Fanuc KAREL source: ko00053.KL

-- PROVISIONAL review KL for V1013-1; original PC SHA256 1e71e2e0424b7fda3cae7a66e169d6796f6002b1d3d6ba8bf153a4db3ede6087
-- Incomplete behavior may be omitted. Consult companion uncertainty JSON. Do not deploy.
PROGRAM KO00053
%NOLOCKGROUP
BEGIN
  -- UNRESOLVED_PC offsets 5-12; opcodes 9D,23
  -- UNRESOLVED_PC offsets 17-69; opcodes 27,27,49,7E,AD,27,49,7E,AD,22,31,7E,4A
  -- UNRESOLVED_PC offsets 74-78; opcodes 7F
END KO00053
